FUNCTION FC_AllError : BOOL
VAR_INPUT
	stStatus	:	ST_FSM_Status;
END_VAR
VAR
END_VAR

FC_AllError := (stStatus.stZ1.eStep = E_Z1_Step.NeOrError) OR
                 (stStatus.stZ2.eStep = E_Z2_Step.NeOrError) OR
                 (stStatus.stZ3.eStep = E_Z3_Step.NeOrError) OR	
                 (stStatus.stZ4.eStep = E_Z4_Step.NeOrError) OR
                 (stStatus.stZ5.eStep = E_Z5_Step.NeOrError) OR	
                 (stStatus.stZ6.eStep = E_Z6_Step.NeOrError);

END_FUNCTION

(* stored: Version 1.1.0.1
   POU FC_AllError: Id {baad097d-0e52-0087-0378-5474cb8c6d28}, SpecialFunc None *)
